FUNCTION_BLOCK fb_ejector_io
VAR_IN_OUT
	var_ref_vac : ref_eje_io;
END_VAR
VAR_INPUT
	in_flg_run : BOOL;
	in_wire_sensVac : BOOL;
	in_wire_sensBrk : BOOL;
	in_var_breakTime: TIME;
	in_var_timerOut : TIME;
END_VAR
VAR_OUTPUT
	out_flg_run : BOOL;
	out_wire_ejeVac : BOOL;
	out_wire_ejeBrk : BOOL;
END_VAR
VAR
END_VAR

out_flg_run := in_flg_run;

var_ref_vac.input.in_flg_sensVac := in_wire_sensVac;
var_ref_vac.input.in_flg_sensBrk := in_wire_sensBrk;

out_wire_ejeVac := var_ref_vac.output.out_flg_ejeVac;
out_wire_ejeBrk := var_ref_vac.output.out_flg_ejeBrk;

var_ref_vac.param.var_BrkTime := in_var_breakTime;
var_ref_vac.param.var_timeOut := in_var_timerOut;

END_FUNCTION_BLOCK

(* stored: Version 1.1.0.1, ProductVersion 3.1.4024.11
   POU fb_ejector_io: Id {134bb3f7-4894-4147-909a-30a7424396fd}, SpecialFunc None *)
